// TIA Portal V20 export
DATA_BLOCK "DB_Sensor"   // DB22
{ S7_Optimized_Access := 'TRUE' }
// stored: AutoNumber false, MemoryReserve 100
   VAR
      "-----  SILOS  -----" : Bool := FALSE;
   END_VAR
   VAR RETAIN
      "010BX1" { S7_SetPoint := 'True'} : "typeSensor";   // placeholder
   END_VAR
BEGIN
   "010BX1"."name" := WSTRING#'F1';
   "010BX1".signal := TRUE;
   "010BX1".on := TRUE;
   "010BX1".off := TRUE;
   "010BX1".onOff := TRUE;
   "010BX1".onTime := T#10S;
   "010BX1".offTime := T#10S;
   "010BX1".sensorFault := FALSE;
   "010BX1".sensorFaultCounter := 0;
   "010BX1".sensorOnFault := T#1M;
   "010BX1".sensorOffFault := T#1M;
   "010BX1".onMeasuring := 157000.0;
   "010BX1".offMeasuring := 0.0;
   "010BX1".onMeasuringTime := T#2M_37S_254MS;
   "010BX1".offMeasuringTime := T#0MS;
   "010BX1".onMeasuringLast := 0.0;
   "010BX1".offMeasuringLast := 0.0;
   "010BX1".onMeasuringLastTime := T#153MS;
   "010BX1".offMeasuringLastTime := T#376MS;
   "010BX1".color := 1;
   "010BX1".colorFiltered := 1;
   "010BX1".distanceTravelled := 1000;
   "010BX1".force := FALSE;
   "010BX1".forceOn := FALSE;
   "010BX1".forceOff := FALSE;
END_DATA_BLOCK
